// TIA Portal project "Rowerzysta" (V14)

(* hardware
DEVICE "S7-1200 station_1"  S7-1200 Station
   slot 0: "Rack_0"  S7-1200 Rack  Rack  V1.0
   slot 1: "PLC_1"  Unspecific CPU 1200  6ES7 2XX-XXXXX-XXXX  V4.2
*)

// ===== PLC "PLC_1"  Unspecific CPU 1200 =====

VAR_GLOBAL   // PLC tag table "Default tag table"
   "zacznij_liczyc" AT %M20.0 : Bool;
   "start!" AT %M20.1 : Bool;
   "stop!" AT %M20.2 : Bool;
   "wykonana_praca" AT %MD12 : Real;
   "max_pracy_rowerzysty" AT %MD0 : Real;
   "potencjometr" AT %ID64 : Real;
   "za_ile_zejde" AT %MD50 : Time;
END_VAR

DATA_BLOCK "Rowerzysta_DB"   // DB1
{ S7_Optimized_Access := 'TRUE' }
VERSION : 0.1
// stored: InstanceOfName Rowerzysta
"Rowerzysta"
BEGIN
END_DATA_BLOCK

FUNCTION_BLOCK "Rowerzysta"   // FB1, SCL
{ S7_Optimized_Access := 'TRUE' }
VERSION : 0.1
   VAR_INPUT
      aktualna_moc : Real;
      czas_przerwania : Time;
      max_pracy_jaki_jestes_w_stanie_wykonac : Real;
   END_VAR
   VAR_OUTPUT
      w_tym_tempie_zejdziesz_za : Time;
      nie_dam_rady : Bool;
   END_VAR
   VAR_IN_OUT
      przepedalowana_praca : Real;
   END_VAR
   VAR
      wartosc_poprzednia : Real;
      praca_chwilowa : Real;
   END_VAR
BEGIN
   #nie_dam_rady := #przepedalowana_praca > #max_pracy_jaki_jestes_w_stanie_wykonac;
   IF NOT #nie_dam_rady THEN
       #praca_chwilowa := (#wartosc_poprzednia + #aktualna_moc) * 0.5 * T_CONV(#czas_przerwania);
       #przepedalowana_praca := #przepedalowana_praca + #praca_chwilowa;
       #w_tym_tempie_zejdziesz_za := T_CONV(REAL_TO_DINT((#max_pracy_jaki_jestes_w_stanie_wykonac - #przepedalowana_praca) / #aktualna_moc));
       #wartosc_poprzednia := #aktualna_moc;
   ELSE
       #w_tym_tempie_zejdziesz_za := T_CONV(0);
       #nie_dam_rady := TRUE;
   END_IF;
END_FUNCTION_BLOCK

ORGANIZATION_BLOCK "Main"   // OB1, LAD, ProgramCycle
TITLE = "Main Program Sweep (Cycle)"
{ S7_Optimized_Access := 'TRUE' }
VERSION : 0.1
   VAR_INPUT
      Initial_Call : Bool;   // Initial call of this OB
      Remanence : Bool;   // =True, if remanent data are available
   END_VAR
   VAR_TEMP   // added for the SCL form of the ladder/FBD networks
      _w1 : Bool;
      _w2 : Bool;
   END_VAR
BEGIN

REGION Network 1
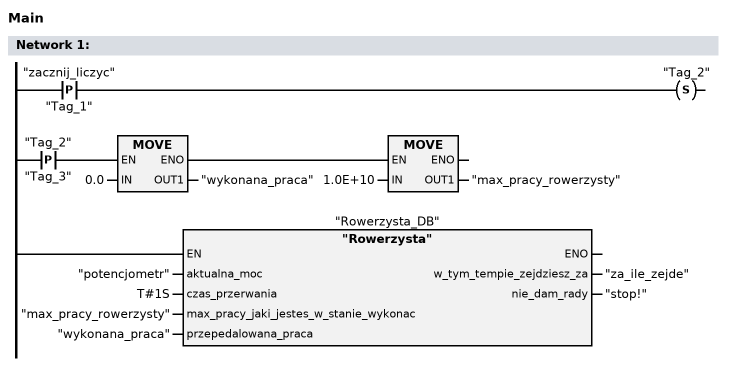
   RUNG wire#powerrail
      P_Contact(operand := "zacznij_liczyc", bit := "Tag_1")
      S_Coil( "Tag_2" )
   END_RUNG
   RUNG wire#powerrail
      P_Contact(operand := "Tag_2", bit := "Tag_3")
      Move(in := 0.0, out1 => "wykonana_praca")
      Move(in := 1.0E+10, out1 => "max_pracy_rowerzysty")
   END_RUNG
   RUNG wire#powerrail
      "Rowerzysta_DB"(aktualna_moc := "potencjometr", czas_przerwania := T#1S, max_pracy_jaki_jestes_w_stanie_wykonac := "max_pracy_rowerzysty", przepedalowana_praca := "wykonana_praca", w_tym_tempie_zejdziesz_za => "za_ile_zejde", nie_dam_rady => "stop!")
   END_RUNG
   // the same network as SCL:
   #_w1 := "zacznij_liczyc" AND NOT "Tag_1";   // rising edge of "zacznij_liczyc"
   "Tag_1" := "zacznij_liczyc";
   IF #_w1 THEN "Tag_2" := TRUE; END_IF;
   #_w2 := "Tag_2" AND NOT "Tag_3";   // rising edge of "Tag_2"
   "Tag_3" := "Tag_2";
   IF #_w2 THEN
       "wykonana_praca" := 0.0;
       "max_pracy_rowerzysty" := 1.0E+10;
   END_IF;
   "Rowerzysta_DB"(aktualna_moc := "potencjometr",   // "Rowerzysta"
                   czas_przerwania := T#1S,
                   max_pracy_jaki_jestes_w_stanie_wykonac := "max_pracy_rowerzysty",
                   przepedalowana_praca := "wykonana_praca",
                   w_tym_tempie_zejdziesz_za => "za_ile_zejde",
                   nie_dam_rady => "stop!");
END_REGION
END_ORGANIZATION_BLOCK